// TIA Portal V19 export
FUNCTION "CallLsntpServer" : Void   // FC1, LAD
// stored: SetENOAutomatically false
   VAR_IN_OUT
      instLSNTP_Server : "LSNTP_Server";
   END_VAR
BEGIN

REGION Network 1
   // With the LSNTP_Server block, the NTP server will be enabled on S7 PLC, to wich the NTP client (e.g. Panel), can synchronize their data and time.
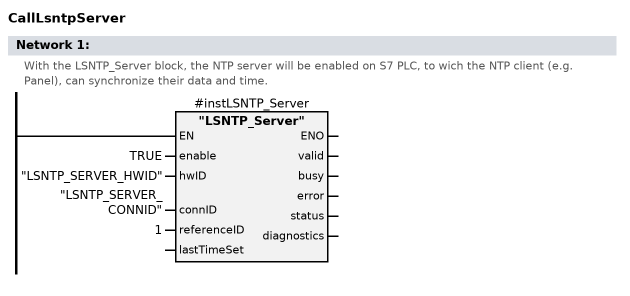
   RUNG wire#powerrail
      #instLSNTP_Server(enable := TRUE, hwID := "LSNTP_SERVER_HWID", connID := "LSNTP_SERVER_CONNID", referenceID := 1, lastTimeSet :=, valid =>, busy =>, error =>, status =>, diagnostics =>)
   END_RUNG
   // the same network as SCL:
   #instLSNTP_Server(enable := TRUE,   // "LSNTP_Server"
                     hwID := "LSNTP_SERVER_HWID",
                     connID := "LSNTP_SERVER_CONNID",
                     referenceID := 1);
END_REGION
END_FUNCTION
